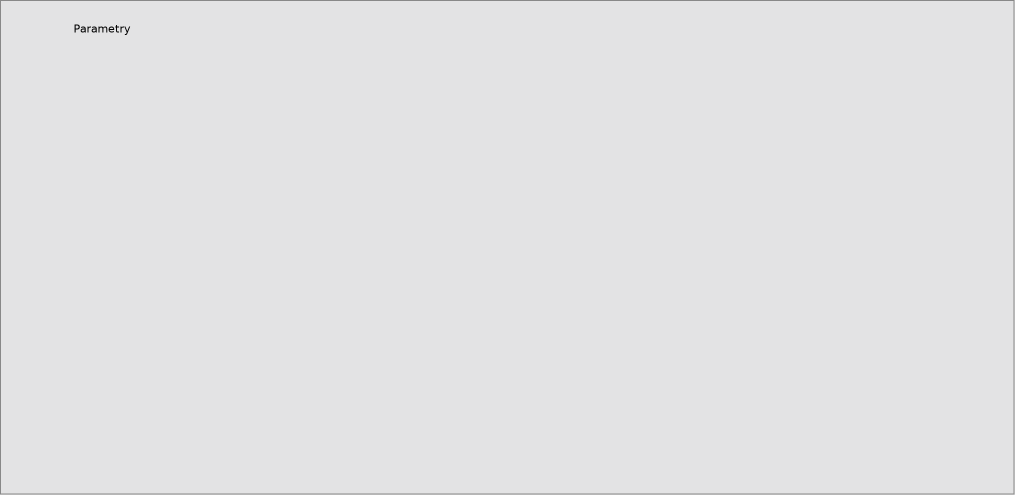
VISUALIZATION F_01_Parameters  // 1015x495
VAR_IN_OUT
	stScreenData	: ST_MCHMIPrepareScreen_01_XX;
	
END_VAR
    Label (27,14 150x30), "Parametry"
END_VISUALIZATION

(* stored: Version 1.1.0.1
   Visu F_01_Parameters: Id {ed0202d9-4538-0fab-0acd-486678a23665} *)
